FUNCTION_BLOCK FB_DcPump EXTENDS FB_ComponentBase IMPLEMENTS I_Pump
VAR
	_InSimulation : BOOL;
END_VAR

//{warning 'Add method implementation '}
METHOD CyclicLogic
IF _InSimulation THEN
	CyclicSimulate();
ELSE
	;
END_IF
END_METHOD

METHOD CyclicSimulate
VAR_INPUT
	flow : INT;
END_VAR
END_METHOD

PROPERTY InSimulation : BOOL
GET
InSimulation := _InSimulation;
END_GET
SET
_InSimulation := InSimulation;
END_SET
END_PROPERTY

{warning 'Add property implementation'}
PROPERTY Speed : LREAL
GET
END_GET
SET
END_SET
END_PROPERTY

{warning 'Add method implementation '}
METHOD Start : BOOL
END_METHOD

{warning 'Add method implementation '}
METHOD Stop
END_METHOD

END_FUNCTION_BLOCK

(* stored: Version 1.1.0.1
   POU FB_DcPump: Id {3d499173-4467-460c-ad21-fdc72eed9e4f}, SpecialFunc None
   Method CyclicLogic: Id {2cb5250d-3879-433b-85a1-ffc3b0b198de}
   Method CyclicSimulate: Id {02bba3ba-972d-4462-aa8d-f4c05e2edc4c}
   Property InSimulation: Id {dfdb7749-1423-400d-a406-fd150c39b8f2}
   Get Get: Id {df2ad642-6298-4388-ad6e-24011b4c836b}
   Set Set: Id {bf531ac0-8964-4647-866d-67bd1fb0539d}
   Property Speed: Id {cee3d3c6-e803-4f41-941f-1a84ad0d5631}
   Get Get: Id {6790faf5-0d5b-4725-aa5c-6b8479fe6589}
   Set Set: Id {d9462662-6bf3-4fb8-95ed-5fef9f0d7807}
   Method Start: Id {eaaab0dd-99dd-42ee-ba88-41b5070224a8}
   Method Stop: Id {6fffd754-8270-49f2-8cd1-eb16cf6c7adb} *)
